(* CoDeSys 2.3.8.0 project: BC9000.pr6 *)
(* Libraries: STANDARD.LB6 5.6.98 11:03:02 *)

(* POU MAIN, ST *)
PROGRAM MAIN
VAR
(*Zmienne, ktore nie zostana utracone*)
	Persistant_Bool AT %MX0.0:	BOOL;	(*1 bit w bajcie 0*)
	Persistant_Integer AT %MB2:	INT;		(*2 bajty*)
	Persistant_Word AT %MB4:		WORD;	(*2 bajty*)
	Persistant_String AT %MB6:		STRING(9);(*Zmienna typu string ograniczona do 9 bajtow*)
	Persistant_Byte AT %MB16:		BYTE;	(*2 bajty*)
	Persistant_Real AT %MB18:	REAL; 	(*4 bajty*)
(*Zmienne, ktore zostana utracone po zaladowaniu nowego programu*)
	Remanent_Bool AT %MX100.0:	BOOL;	(*1 bit w bajcie 100*)
	Remanent_Integer AT %MB102:	INT;		(*2 bajty*)
	Remanent_Word AT %MB104:	WORD;	(*2 bajty*)
	Remanent_String AT %MB106:	STRING(9);(*Zmienna typu string ograniczona do 9 bajtow*)
	Remanent_Byte AT %MB116:	BYTE;	(*2 bajty*)
	Remanent_Real AT %MB118:	REAL; 	(*4 bajty*)
END_VAR
;
END_PROGRAM
